PROGRAM MAIN
VAR
	Ialive : Int;
END_VAR

Ialive := Ialive + 1;

END_PROGRAM

(* stored: Version 1.1.0.1
   POU MAIN: Id {e6db5317-5b9c-486b-bde3-90f98110c465}, SpecialFunc None *)
